{attribute 'qualified_only'}
{attribute 'strict'}
TYPE AxisBufferMode :
(
	Aborting := MC_Aborting,
	Buffered := MC_Buffered,
	BlendingLow := MC_BlendingLow,
	BlendingPrevious := MC_BlendingPrevious,
	BlendingNext := MC_BlendingNext,
	BlendingHigh := MC_BlendingHigh
) UINT;
END_TYPE

(* stored: Version 1.1.0.1, ProductVersion 3.1.4024.12
   DUT AxisBufferMode: Id {eedb7269-49ec-07a7-15dc-a47e35097a7b} *)
